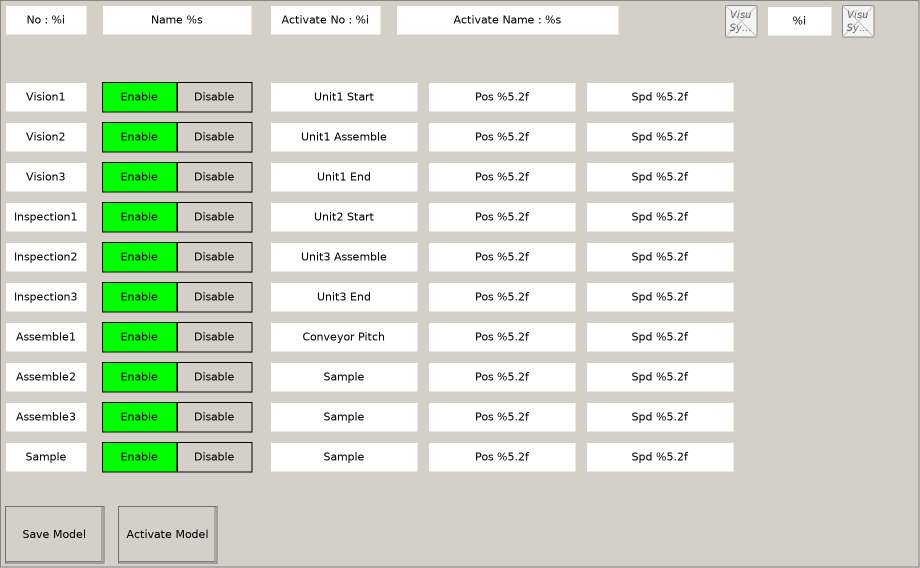
VISUALIZATION Model  // 920x568
    Textfield (102,5 150x30), "Name %s", text variable: astInputModel[iModelIndex].sName
        OnMouseClick: write the text variable via Edit
    Textfield (5,5 82x30), "No : %i", text variable: astInputModel[iModelIndex].iNumber
    Image (725,5 32x32), invisible if: bInvisibleLeft, image: VisuSymbols.Symbols.ArrowBoldLeft
        OnMouseClick: execute { iModelindex := iModelindex -1; }
    Image (842,5 32x32), invisible if: bInvisibleRight, image: VisuSymbols.Symbols.ArrowBoldRight
        OnMouseClick: execute { iModelindex := iModelindex +1; }
    Textfield (767,6 65x30), "%i", text variable: astInputModel[iModelIndex].iNumber
        OnMouseClick: write iModelIndex via Default, min 1, max cMaxModelNo
    Textfield (5,82 82x30), "Vision1"
    Rectangle (102,82 75x30), "Enable", colour toggle: astInputModel[iModelIndex].abType[1]
        OnMouseClick: execute { astInputModel[iModelIndex].abType[1] := FALSE; }
    Rectangle (177,82 75x30), "Disable", colour toggle: astInputModel[iModelIndex].abType[1]
        OnMouseClick: execute { astInputModel[iModelIndex].abType[1] := true; }
    Textfield (5,122 82x30), "Vision2"
    Rectangle (102,122 75x30), "Enable", colour toggle: astInputModel[iModelIndex].abType[2]
        OnMouseClick: execute { astInputModel[iModelIndex].abType[2] := FALSE; }
    Rectangle (177,122 75x30), "Disable", colour toggle: astInputModel[iModelIndex].abType[2]
        OnMouseClick: execute { astInputModel[iModelIndex].abType[2] := true; }
    Textfield (5,162 82x30), "Vision3"
    Rectangle (102,162 75x30), "Enable", colour toggle: astInputModel[iModelIndex].abType[3]
        OnMouseClick: execute { astInputModel[iModelIndex].abType[3] := FALSE; }
    Rectangle (177,162 75x30), "Disable", colour toggle: astInputModel[iModelIndex].abType[3]
        OnMouseClick: execute { astInputModel[iModelIndex].abType[3] := true; }
    Textfield (5,202 82x30), "Inspection1"
    Rectangle (102,202 75x30), "Enable", colour toggle: astInputModel[iModelIndex].abType[4]
        OnMouseClick: execute { astInputModel[iModelIndex].abType[4] := FALSE; }
    Rectangle (177,202 75x30), "Disable", colour toggle: astInputModel[iModelIndex].abType[4]
        OnMouseClick: execute { astInputModel[iModelIndex].abType[4] := true; }
    Textfield (5,242 82x30), "Inspection2"
    Rectangle (102,242 75x30), "Enable", colour toggle: astInputModel[iModelIndex].abType[5]
        OnMouseClick: execute { astInputModel[iModelIndex].abType[5] := FALSE; }
    Rectangle (177,242 75x30), "Disable", colour toggle: astInputModel[iModelIndex].abType[5]
        OnMouseClick: execute { astInputModel[iModelIndex].abType[5] := true; }
    Textfield (5,282 82x30), "Inspection3"
    Rectangle (102,282 75x30), "Enable", colour toggle: astInputModel[iModelIndex].abType[6]
        OnMouseClick: execute { astInputModel[iModelIndex].abType[6] := FALSE; }
    Rectangle (177,282 75x30), "Disable", colour toggle: astInputModel[iModelIndex].abType[6]
        OnMouseClick: execute { astInputModel[iModelIndex].abType[6] := true; }
    Textfield (5,322 82x30), "Assemble1"
    Rectangle (102,322 75x30), "Enable", colour toggle: astInputModel[iModelIndex].abType[7]
        OnMouseClick: execute { astInputModel[iModelIndex].abType[7] := FALSE; }
    Rectangle (177,322 75x30), "Disable", colour toggle: astInputModel[iModelIndex].abType[7]
        OnMouseClick: execute { astInputModel[iModelIndex].abType[7] := true; }
    Textfield (5,362 82x30), "Assemble2"
    Rectangle (102,362 75x30), "Enable", colour toggle: astInputModel[iModelIndex].abType[8]
        OnMouseClick: execute { astInputModel[iModelIndex].abType[8] := FALSE; }
    Rectangle (177,362 75x30), "Disable", colour toggle: astInputModel[iModelIndex].abType[8]
        OnMouseClick: execute { astInputModel[iModelIndex].abType[8] := true; }
    Textfield (5,402 82x30), "Assemble3"
    Rectangle (102,402 75x30), "Enable", colour toggle: astInputModel[iModelIndex].abType[9]
        OnMouseClick: execute { astInputModel[iModelIndex].abType[9] := FALSE; }
    Rectangle (177,402 75x30), "Disable", colour toggle: astInputModel[iModelIndex].abType[9]
        OnMouseClick: execute { astInputModel[iModelIndex].abType[9] := true; }
    Textfield (5,442 82x30), "Sample"
    Rectangle (102,442 75x30), "Enable", colour toggle: astInputModel[iModelIndex].abType[10]
        OnMouseClick: execute { astInputModel[iModelIndex].abType[10] := FALSE; }
    Rectangle (177,442 75x30), "Disable", colour toggle: astInputModel[iModelIndex].abType[10]
        OnMouseClick: execute { astInputModel[iModelIndex].abType[10] := true; }
    Button (5,506 99x57), "Save Model", colour toggle: bLpSaveModelData
        tap bBtSaveModelData
    Button (118,506 99x57), "Activate Model", colour toggle: bLpActivateModel
        tap bBtActivateModel
    Textfield (396,5 223x30), "Activate Name : %s", text variable: stCurrnetModel.sName
        OnMouseClick: write the text variable via Edit
    Textfield (270,5 111x30), "Activate No : %i", text variable: stCurrnetModel.iNumber
    Group (270,82 148x390)
        Textfield (0,0 148x30), "Unit1 Start"
        Textfield (0,40 148x30), "Unit1 Assemble"
        Textfield (0,80 148x30), "Unit1 End"
        Textfield (0,120 148x30), "Unit2 Start"
        Textfield (0,160 148x30), "Unit3 Assemble"
        Textfield (0,200 148x30), "Unit3 End"
        Textfield (0,240 148x30), "Conveyor Pitch"
        Textfield (0,280 148x30), "Sample"
        Textfield (0,320 148x30), "Sample"
        Textfield (0,360 148x30), "Sample"
    Textfield (428,82 148x30), "Pos %5.2f", text variable: astInputModel[iModelindex].arPosition[1]
        OnMouseClick: write the text variable via Default
    Textfield (428,122 148x30), "Pos %5.2f", text variable: astInputModel[iModelindex].arPosition[2]
        OnMouseClick: write the text variable via Default
    Textfield (428,162 148x30), "Pos %5.2f", text variable: astInputModel[iModelindex].arPosition[3]
        OnMouseClick: write the text variable via Default
    Textfield (428,202 148x30), "Pos %5.2f", text variable: astInputModel[iModelindex].arPosition[4]
        OnMouseClick: write the text variable via Default
    Textfield (428,242 148x30), "Pos %5.2f", text variable: astInputModel[iModelindex].arPosition[5]
        OnMouseClick: write the text variable via Default
    Textfield (428,282 148x30), "Pos %5.2f", text variable: astInputModel[iModelindex].arPosition[6]
        OnMouseClick: write the text variable via Default
    Textfield (428,322 148x30), "Pos %5.2f", text variable: astInputModel[iModelindex].arPosition[7]
        OnMouseClick: write the text variable via Default
    Textfield (428,362 148x30), "Pos %5.2f", text variable: astInputModel[iModelindex].arPosition[8]
        OnMouseClick: write the text variable via Default
    Textfield (428,402 148x30), "Pos %5.2f", text variable: astInputModel[iModelindex].arPosition[9]
        OnMouseClick: write the text variable via Default
    Textfield (428,442 148x30), "Pos %5.2f", text variable: astInputModel[iModelindex].arPosition[10]
        OnMouseClick: write the text variable via Default
    Textfield (586,82 148x30), "Spd %5.2f", text variable: astInputModel[iModelindex].arSpeed[1]
        OnMouseClick: write the text variable via Default
    Textfield (586,122 148x30), "Spd %5.2f", text variable: astInputModel[iModelindex].arSpeed[2]
        OnMouseClick: write the text variable via Default
    Textfield (586,162 148x30), "Spd %5.2f", text variable: astInputModel[iModelindex].arSpeed[3]
        OnMouseClick: write the text variable via Default
    Textfield (586,202 148x30), "Spd %5.2f", text variable: astInputModel[iModelindex].arSpeed[4]
        OnMouseClick: write the text variable via Default
    Textfield (586,242 148x30), "Spd %5.2f", text variable: astInputModel[iModelindex].arSpeed[5]
        OnMouseClick: write the text variable via Default
    Textfield (586,282 148x30), "Spd %5.2f", text variable: astInputModel[iModelindex].arSpeed[6]
        OnMouseClick: write the text variable via Default
    Textfield (586,322 148x30), "Spd %5.2f", text variable: astInputModel[iModelindex].arSpeed[7]
        OnMouseClick: write the text variable via Default
    Textfield (586,362 148x30), "Spd %5.2f", text variable: astInputModel[iModelindex].arSpeed[8]
        OnMouseClick: write the text variable via Default
    Textfield (586,402 148x30), "Spd %5.2f", text variable: astInputModel[iModelindex].arSpeed[9]
        OnMouseClick: write the text variable via Default
    Textfield (586,442 148x30), "Spd %5.2f", text variable: astInputModel[iModelindex].arSpeed[10]
        OnMouseClick: write the text variable via Default
END_VISUALIZATION

(* stored: Version 1.1.0.1
   Visu Model: Id {1ad760d6-49f5-452c-b8f8-8c412b5e472d} *)
